(* IEC 61131-3 sources: Industry-PLC-LLM/data/PLCBEAD_repo/PLCBEAD_PLCEmbed-main/PLC-BEAD/Source/GEB/F_POWER, 1 file *)

(* ---- F_POWER.ST ---- *)
FUNCTION F_POWER:REAL
	VAR_INPUT
		A :	REAL;
		X :	REAL;
		N :	REAL;
	END_VAR

	F_POWER := A * EXPT(X,N);
END_FUNCTION

PROGRAM program0
  VAR
    LocalVar0 : REAL;
	LocalVaR1  : REAL;
	LocalVaR2 : REAL;
	  LocalOUT  : REAL;
  END_VAR
  	LocalOUT := F_POWER(LocalVar0, LocalVaR1 , LocalVaR2);
END_PROGRAM
